// TwinCAT 3 PLC project basicFunsPlc
// ProgramVersion: 3.1.4024.0
// libraries:
//   Tc2_Standard, * (Beckhoff Automation GmbH)
//   Tc2_System, * (Beckhoff Automation GmbH)
//   Tc3_Module, * (Beckhoff Automation GmbH)
// project tree:
//   / PlcTask.TcTTO
//   POUs/ MAIN.TcPOU
// real-time tasks:
//   TASK PlcTask: cycle T#10ms, priority 20, ADS port 350

CONFIGURATION basicFunsPlc
    RESOURCE PLC ON TwinCAT3
        TASK PlcTask(INTERVAL := T#10ms, PRIORITY := 20);
        PROGRAM MAIN WITH PlcTask : MAIN;
    END_RESOURCE
END_CONFIGURATION

// ---- POUs/MAIN.TcPOU
PROGRAM MAIN
VAR
	//fbTof : TOF := (PT := T#10S);
	fbTrig : R_TRIG;
	bBool : BOOL;
	trigCounter : ULINT;
END_VAR

//fbTof(IN := bBool);
fbTrig(CLK := bBool);
IF fbTrig.Q THEN
	trigCounter := trigCounter + 1;
END_IF

END_PROGRAM
